TYPE Read_BLVac2_Values_To_PC_Struct :
UNION
	S_BLVac2Values_To_PC:S_BLVac2Values_To_PC_Struct;
END_UNION
END_TYPE

(* stored: Version 1.1.0.1, ProductVersion 3.1.4024.16
   DUT Read_BLVac2_Values_To_PC_Struct: Id {b8667341-b475-4af0-b572-1c68f5c63061} *)
